FUNCTION_BLOCK Player
VAR
	iScoreValue :INT;
	sName : STRING;	

END_VAR

PROPERTY Name : STRING
GET
Name := sName;
END_GET
SET
sName := Name;
END_SET
END_PROPERTY

PROPERTY Score : INT
GET
Score := iScoreValue;
END_GET
SET
iScoreValue := Score;
END_SET
END_PROPERTY

END_FUNCTION_BLOCK

(* stored: Version 1.1.0.1, ProductVersion 3.1.4024.12
   POU Player: Id {be859fcf-6167-4c07-bf0f-51afc398156f}, SpecialFunc None
   Property Name: Id {64974a64-178c-4793-a0f3-4c0ca1a98da7}
   Get Get: Id {f1ccf210-f8f6-417c-8f98-8591785ea4e9}
   Set Set: Id {bd4aff2d-4ae1-434c-9305-4632005107cb}
   Property Score: Id {e90bf12a-d274-4271-8ed9-9cfba22a2b3a}
   Get Get: Id {aff5a276-3177-4421-8dd8-8c0d4affd5db}
   Set Set: Id {2d372158-335c-4cc0-b4e6-0630bcda2b1e} *)
